(* CODESYS project io.library
   Company: MyCompany AB
   DefaultNamespace: IO
   Version: 0.1.0.1
   Placeholder: Inputs and Outputs
   Author: Milan Cic
   Description: This library holds functionality for testing
   Title: Inputs and Outputs

Project tree, tasks and I/O mapping:
  libraries: Tc2_Standard, * (Beckhoff Automation GmbH); Tc2_System, * (Beckhoff Automation GmbH); Tc3_Module, * (Beckhoff Automation GmbH)
  DUTs/
  GVLs/
  POUs/
    function block FB_CalcAdder [ST]
  Version/
    global variables Global_Version
*)

// Version/Global_Version
{attribute 'TcGenerated'}
{attribute 'no-analysis'}
{attribute 'linkalways'}
// This function has been automatically generated from the project information.
VAR_GLOBAL CONSTANT
	{attribute 'const_non_replaced'}
	stLibVersion_Inputs_and_Outputs : ST_LibVersion := (iMajor := 0, iMinor := 1, iBuild := 0, iRevision := 1, nFlags := 0, sVersion := '0.1.0.1');
END_VAR

// POUs/FB_CalcAdder
FUNCTION_BLOCK FB_CalcAdder
VAR_INPUT
	firstVar	:	INT;
	secondVar	:	INT;
END_VAR
VAR_OUTPUT
	result		:	int;
END_VAR
VAR
END_VAR

result	:=	firstVar +	secondVar + 3;

END_FUNCTION_BLOCK
